(* Logix 5000 project; controller PRU vendor 1 type 14 code 107 rev 20.13; software revision 20.01; part 9 of 17 *)
(* tags used below, declared in another part *)
   AFI : BOOL;
   COOL_FOR_MOTOR_STOP : BOOL;
   CR0_CON1_HTR1_GON : BOOL;   // ZONE 1 (L1,L2,L3)
   CR0_CON1_HTR1_LON : BOOL;   // AUTO LOGIC - ZONE 1 HEATER CONTACTOR
   CR1_CON2_HTR2_GON : BOOL;   // ZONE 2 (L1,L2,L3)
   CR1_CON2_HTR2_LON : BOOL;   // AUTO LOGIC - ZONE 2 HEATER CONTACTOR
   CR2_CON3_HTR3_GON : BOOL;   // ZONE 3 (L1,L2,L3)
   CR2_CON3_HTR3_LON : BOOL;   // AUTO LOGIC - ZONE 3 HEATER CONTACTOR
   CR3_CON4_HTR4_GON : BOOL;   // ZONE 4 (L1) ZONE 5 (L2) ZONE 6 (L3)
   CR3_CON4_HTR4_LON : BOOL;   // AUTO LOGIC - ZONES 4-6 HEATER CONTACTOR
   CR4_CON5_HTR5_GON : BOOL;   // ZONE 7 (L1) ZONE 8 (L2) ZONE 9 (L3)
   CR4_CON5_HTR5_LON : BOOL;   // AUTO LOGIC - ZONES 7-9 HEATER CONTACTOR
   CYCLE_ION_DELAY1_TON : TIMER;
   CYCLE_ION_DELAY2_TON : TIMER;
   CYCLE_ION_DELAY3_TON : TIMER;
   CYCLE_ION_DELAY4_TON : TIMER;
   CYCLE_START_ONS : BOOL;
   CYCLE_START_SS : BOOL;   // Begin temperature ramp and hold heat cycle.
   FAULT : DINT[100];
   FAULT_TIMER : TIMER[10000];
   FAULTS_FA6_IOK : BOOL;   // HEATER FAULTS ARE OK.
   FAULTS_FA6A_IOK : BOOL;
   FAULTS_FA6B_IOK : BOOL;
   HEATER_1_ALARM_ION : BOOL;
   HEATER_2_ALARM_ION : BOOL;
   HEATER_3_ALARM_ION : BOOL;
   HEATER_4_ALARM_ION : BOOL;
   HEATER_5_ALARM_ION : BOOL;
   HEATER_FAULTS_IOK : BOOL;   // FA1, FA4, FA6
   HEATERS_CYCLE_ION : BOOL;   // Heaters are commanded on.
   HMI_ALARM_RESET : BOOL;
   HMI_CYCLE_STOP_PB_ION : BOOL;
   HMI_HEATER_START_PB_ION : BOOL;
   HMI_SEQ_1_FINAL_SETPOINT : DINT;
   HMI_SEQ_1_HOLD_TIME : DINT;
   HMI_SEQ_1_RATE : DINT;
   HMI_SEQ_2_FINAL_SETPOINT : DINT;
   HMI_SEQ_2_HOLD_TIME : DINT;
   HMI_SEQ_2_RATE : DINT;
   HMI_SEQ_3_FINAL_SETPOINT : DINT;
   HMI_SEQ_3_HOLD_TIME : DINT;
   HMI_SEQ_3_RATE : DINT;
   HMI_ZONE1_FINAL_SETPOINT : REAL;
   HMI_ZONE2_FINAL_SETPOINT : DINT;
   HMI_ZONE3_FINAL_SETPOINT : DINT;
   HMI_ZONE4_FINAL_SETPOINT : DINT;
   HMI_ZONE5_FINAL_SETPOINT : REAL;
   HMI_ZONE6_FINAL_SETPOINT : REAL;
   HMI_ZONE7_FINAL_SETPOINT : DINT;
   HMI_ZONE8_FINAL_SETPOINT : DINT;
   HMI_ZONE9_FINAL_SETPOINT : DINT;
   ONE_SEC_SS : BOOL;
   PID_ZONE_1_SETPOINT : DINT;
   PID_ZONE_2_SETPOINT : DINT;
   PID_ZONE_3_SETPOINT : DINT;
   PID_ZONE_4_SETPOINT : DINT;
   PID_ZONE_5_SETPOINT : REAL;
   PID_ZONE_6_SETPOINT : REAL;
   PID_ZONE_7_SETPOINT : DINT;
   PID_ZONE_8_SETPOINT : DINT;
   PID_ZONE_9_SETPOINT : DINT;
   PROCESS_SEQUENCER : INT;
   PRODUCTION_ION : BOOL;
   SEQ_1_HOLD_REM : REAL;
   SEQ_1_HOLD_REM_MIN : REAL;
   SEQ_1_HOLD_TIME : DINT;
   SEQ_1_HOLD_TON : TIMER;
   SEQ_1_HOLDING_ION : BOOL;
   SEQ_1_ION : BOOL;
   SEQ_2_HOLD_REM : REAL;
   SEQ_2_HOLD_REM_MIN : REAL;
   SEQ_2_HOLD_TIME : DINT;
   SEQ_2_HOLD_TON : TIMER;
   SEQ_2_HOLDING_ION : BOOL;
   SEQ_2_ION : BOOL;
   SEQ_3_HOLD_REM : REAL;
   SEQ_3_HOLD_REM_MIN : REAL;
   SEQ_3_HOLD_TIME : DINT;
   SEQ_3_HOLD_TON : TIMER;
   SEQ_3_HOLDING_ION : BOOL;
   SEQ_3_ION : BOOL;
   SEQ_RATE : REAL;
   SP_RATIO : REAL;
   SYSTEM_SETPOINT : REAL;
   TE0101 : REAL;
   TE0102 : REAL;
   TE0103 : REAL;
   TE0104 : REAL;
   TE0105 : REAL;
   TE0106 : REAL;
   TE0107 : REAL;
   TE0108 : REAL;
   TE0109 : REAL;
   TE0110 : REAL;
   TE0111 : REAL;
   TE0112 : REAL;
   TE0113 : REAL;
   TE0114 : REAL;
   TE0115 : REAL;
   TE0116 : REAL;
   TE0117 : REAL;
   TE0118 : REAL;
   TE0119 : REAL;
   TE0120 : REAL;
   TE0121 : REAL;
   TE0122 : REAL;
   TE0123 : REAL;
   TE0124 : REAL;
   TEMP_ZONE_1_AVE : REAL;
   TEMPERATURE_SETPOINT_IS_RAMPING : BOOL;
   TEST_VFD_BON : BOOL;
   THRESHOLD : REAL[9000];
   VFD_SHUTDOWN_TEMP : DINT;
   VFDS_BON : BOOL;   // DRYER VFDs HAVE BEEN COMMANDED ON FOR 1 SECOND.
   Z1_L1_AMPS : REAL;
   Z1_L2_AMPS : REAL;
   Z1_L3_AMPS : REAL;
   Z2_L1_AMPS : REAL;
   Z2_L2_AMPS : REAL;
   Z2_L3_AMPS : REAL;
   Z3_L1_AMPS : REAL;
   Z3_L2_AMPS : REAL;
   Z3_L3_AMPS : REAL;
   Z4_L1_AMPS : REAL;
   Z5_L2_AMPS : REAL;
   Z6_L3_AMPS : REAL;
   Z7_L1_AMPS : REAL;
   Z8_L2_AMPS : REAL;
   Z9_L3_AMPS : REAL;
   ZONE_1_TEMP_AVE : DINT;
(* MainProgram, continued *)

ROUTINE B06_FAULTS_FA6_A_HEATER_5800   (* ladder *)
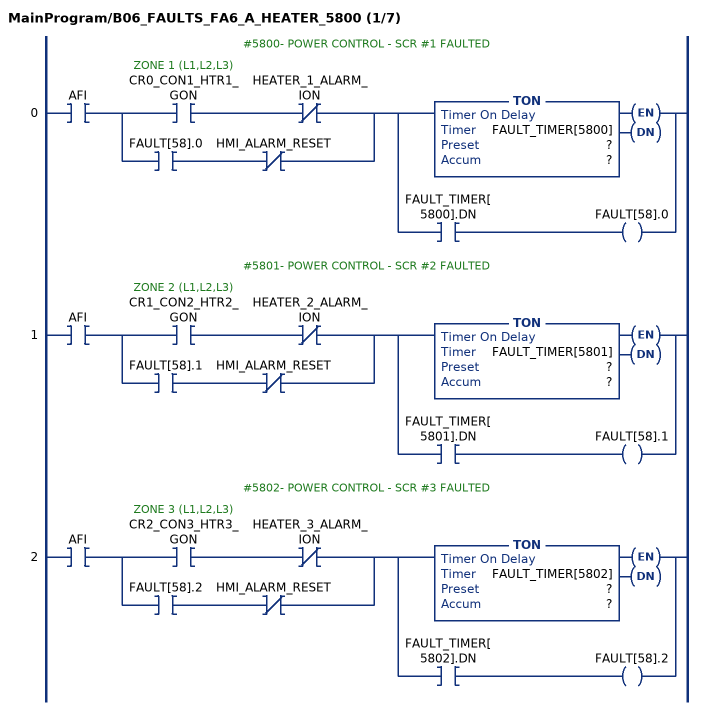
   // #5800- POWER CONTROL - SCR #1 FAULTED
   0: XIC(AFI)[XIC(CR0_CON1_HTR1_GON) XIO(HEATER_1_ALARM_ION) ,XIC(FAULT[58].0) XIO(HMI_ALARM_RESET) ][TON(FAULT_TIMER[5800],?,?) ,XIC(FAULT_TIMER[5800].DN) OTE(FAULT[58].0) ];
   // #5801- POWER CONTROL - SCR #2 FAULTED
   1: XIC(AFI)[XIC(CR1_CON2_HTR2_GON) XIO(HEATER_2_ALARM_ION) ,XIC(FAULT[58].1) XIO(HMI_ALARM_RESET) ][TON(FAULT_TIMER[5801],?,?) ,XIC(FAULT_TIMER[5801].DN) OTE(FAULT[58].1) ];
   // #5802- POWER CONTROL - SCR #3 FAULTED
   2: XIC(AFI)[XIC(CR2_CON3_HTR3_GON) XIO(HEATER_3_ALARM_ION) ,XIC(FAULT[58].2) XIO(HMI_ALARM_RESET) ][TON(FAULT_TIMER[5802],?,?) ,XIC(FAULT_TIMER[5802].DN) OTE(FAULT[58].2) ];
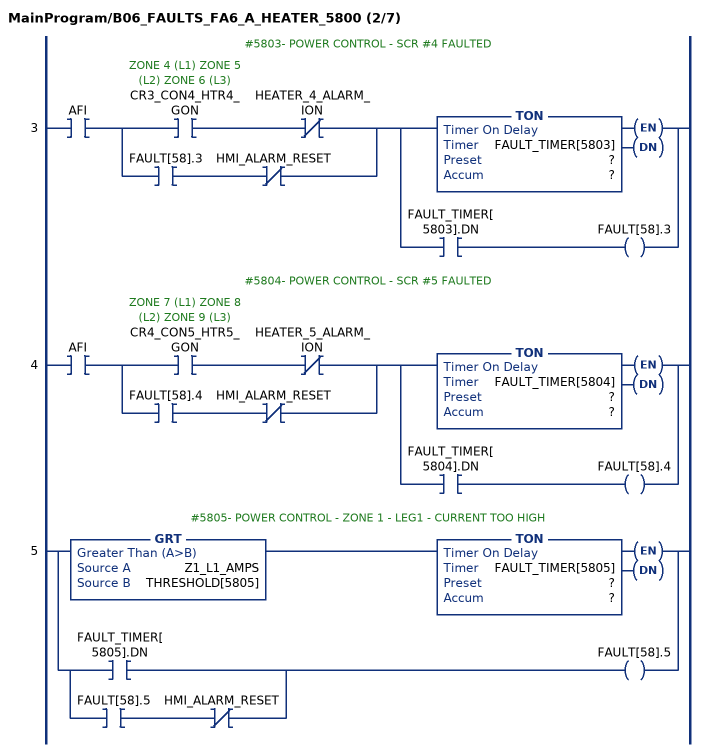
   // #5803- POWER CONTROL - SCR #4 FAULTED
   3: XIC(AFI)[XIC(CR3_CON4_HTR4_GON) XIO(HEATER_4_ALARM_ION) ,XIC(FAULT[58].3) XIO(HMI_ALARM_RESET) ][TON(FAULT_TIMER[5803],?,?) ,XIC(FAULT_TIMER[5803].DN) OTE(FAULT[58].3) ];
   // #5804- POWER CONTROL - SCR #5 FAULTED
   4: XIC(AFI)[XIC(CR4_CON5_HTR5_GON) XIO(HEATER_5_ALARM_ION) ,XIC(FAULT[58].4) XIO(HMI_ALARM_RESET) ][TON(FAULT_TIMER[5804],?,?) ,XIC(FAULT_TIMER[5804].DN) OTE(FAULT[58].4) ];
   // #5805- POWER CONTROL - ZONE 1 - LEG1 - CURRENT TOO HIGH
   5: [GRT(Z1_L1_AMPS,THRESHOLD[5805]) TON(FAULT_TIMER[5805],?,?) ,[XIC(FAULT_TIMER[5805].DN) ,XIC(FAULT[58].5) XIO(HMI_ALARM_RESET) ] OTE(FAULT[58].5) ];
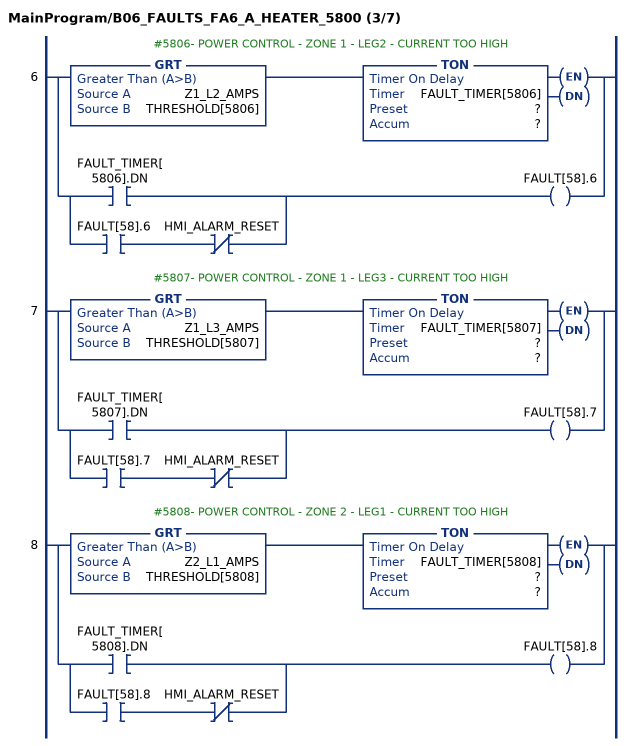
   // #5806- POWER CONTROL - ZONE 1 - LEG2 - CURRENT TOO HIGH
   6: [GRT(Z1_L2_AMPS,THRESHOLD[5806]) TON(FAULT_TIMER[5806],?,?) ,[XIC(FAULT_TIMER[5806].DN) ,XIC(FAULT[58].6) XIO(HMI_ALARM_RESET) ] OTE(FAULT[58].6) ];
   // #5807- POWER CONTROL - ZONE 1 - LEG3 - CURRENT TOO HIGH
   7: [GRT(Z1_L3_AMPS,THRESHOLD[5807]) TON(FAULT_TIMER[5807],?,?) ,[XIC(FAULT_TIMER[5807].DN) ,XIC(FAULT[58].7) XIO(HMI_ALARM_RESET) ] OTE(FAULT[58].7) ];
   // #5808- POWER CONTROL - ZONE 2 - LEG1 - CURRENT TOO HIGH
   8: [GRT(Z2_L1_AMPS,THRESHOLD[5808]) TON(FAULT_TIMER[5808],?,?) ,[XIC(FAULT_TIMER[5808].DN) ,XIC(FAULT[58].8) XIO(HMI_ALARM_RESET) ] OTE(FAULT[58].8) ];
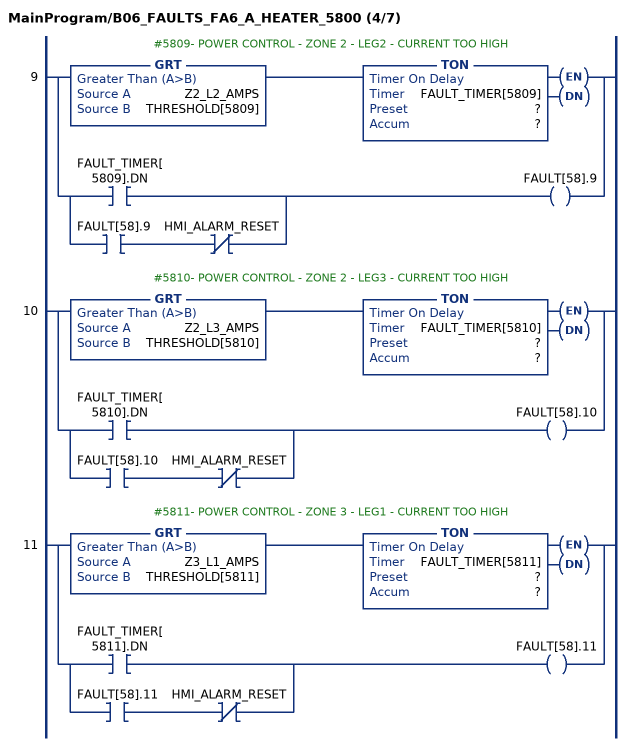
   // #5809- POWER CONTROL - ZONE 2 - LEG2 - CURRENT TOO HIGH
   9: [GRT(Z2_L2_AMPS,THRESHOLD[5809]) TON(FAULT_TIMER[5809],?,?) ,[XIC(FAULT_TIMER[5809].DN) ,XIC(FAULT[58].9) XIO(HMI_ALARM_RESET) ] OTE(FAULT[58].9) ];
   // #5810- POWER CONTROL - ZONE 2 - LEG3 - CURRENT TOO HIGH
   10: [GRT(Z2_L3_AMPS,THRESHOLD[5810]) TON(FAULT_TIMER[5810],?,?) ,[XIC(FAULT_TIMER[5810].DN) ,XIC(FAULT[58].10) XIO(HMI_ALARM_RESET) ] OTE(FAULT[58].10) ];
   // #5811- POWER CONTROL - ZONE 3 - LEG1 - CURRENT TOO HIGH
   11: [GRT(Z3_L1_AMPS,THRESHOLD[5811]) TON(FAULT_TIMER[5811],?,?) ,[XIC(FAULT_TIMER[5811].DN) ,XIC(FAULT[58].11) XIO(HMI_ALARM_RESET) ] OTE(FAULT[58].11) ];
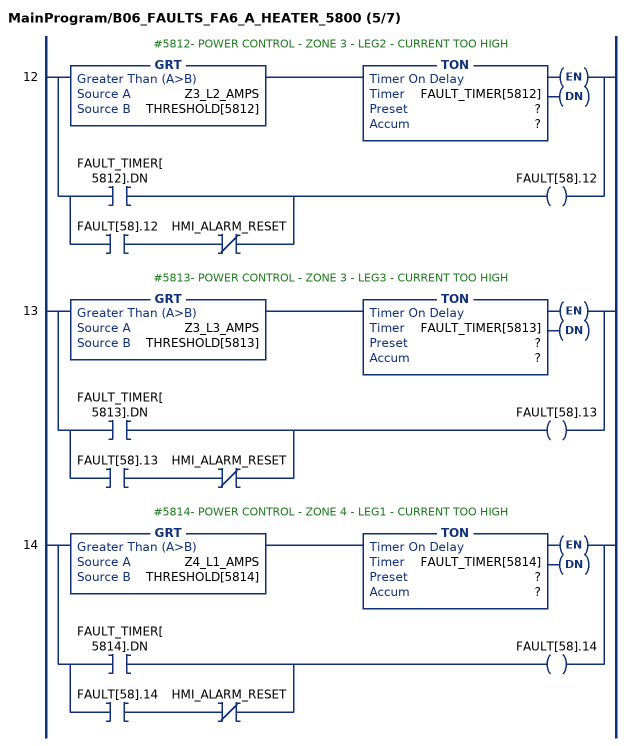
   // #5812- POWER CONTROL - ZONE 3 - LEG2 - CURRENT TOO HIGH
   12: [GRT(Z3_L2_AMPS,THRESHOLD[5812]) TON(FAULT_TIMER[5812],?,?) ,[XIC(FAULT_TIMER[5812].DN) ,XIC(FAULT[58].12) XIO(HMI_ALARM_RESET) ] OTE(FAULT[58].12) ];
   // #5813- POWER CONTROL - ZONE 3 - LEG3 - CURRENT TOO HIGH
   13: [GRT(Z3_L3_AMPS,THRESHOLD[5813]) TON(FAULT_TIMER[5813],?,?) ,[XIC(FAULT_TIMER[5813].DN) ,XIC(FAULT[58].13) XIO(HMI_ALARM_RESET) ] OTE(FAULT[58].13) ];
   // #5814- POWER CONTROL - ZONE 4 - LEG1 - CURRENT TOO HIGH
   14: [GRT(Z4_L1_AMPS,THRESHOLD[5814]) TON(FAULT_TIMER[5814],?,?) ,[XIC(FAULT_TIMER[5814].DN) ,XIC(FAULT[58].14) XIO(HMI_ALARM_RESET) ] OTE(FAULT[58].14) ];
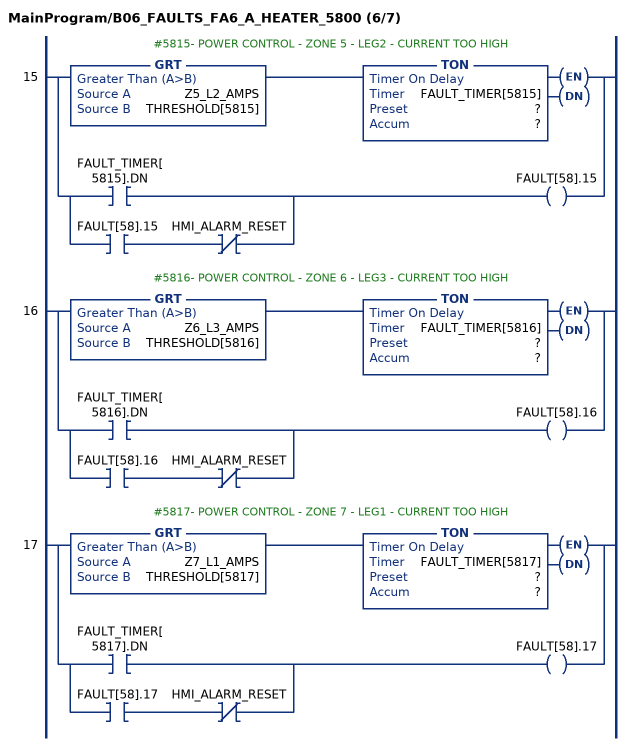
   // #5815- POWER CONTROL - ZONE 5 - LEG2 - CURRENT TOO HIGH
   15: [GRT(Z5_L2_AMPS,THRESHOLD[5815]) TON(FAULT_TIMER[5815],?,?) ,[XIC(FAULT_TIMER[5815].DN) ,XIC(FAULT[58].15) XIO(HMI_ALARM_RESET) ] OTE(FAULT[58].15) ];
   // #5816- POWER CONTROL - ZONE 6 - LEG3 - CURRENT TOO HIGH
   16: [GRT(Z6_L3_AMPS,THRESHOLD[5816]) TON(FAULT_TIMER[5816],?,?) ,[XIC(FAULT_TIMER[5816].DN) ,XIC(FAULT[58].16) XIO(HMI_ALARM_RESET) ] OTE(FAULT[58].16) ];
   // #5817- POWER CONTROL - ZONE 7 - LEG1 - CURRENT TOO HIGH
   17: [GRT(Z7_L1_AMPS,THRESHOLD[5817]) TON(FAULT_TIMER[5817],?,?) ,[XIC(FAULT_TIMER[5817].DN) ,XIC(FAULT[58].17) XIO(HMI_ALARM_RESET) ] OTE(FAULT[58].17) ];
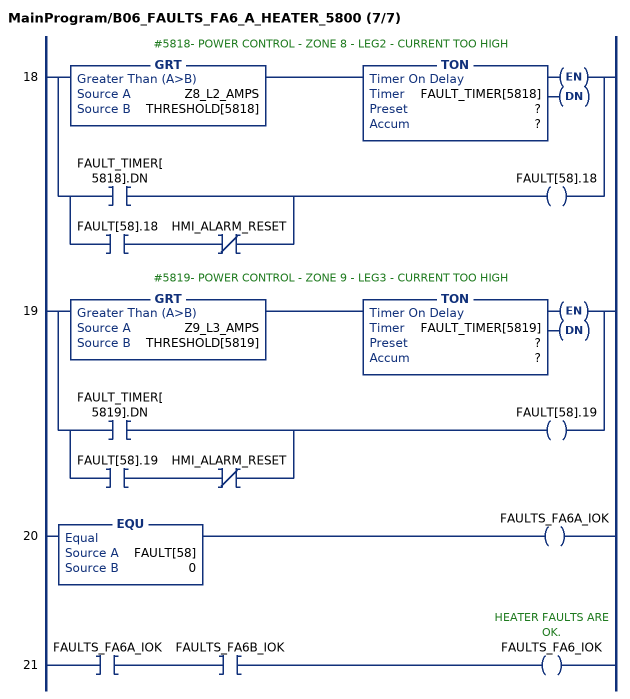
   // #5818- POWER CONTROL - ZONE 8 - LEG2 - CURRENT TOO HIGH
   18: [GRT(Z8_L2_AMPS,THRESHOLD[5818]) TON(FAULT_TIMER[5818],?,?) ,[XIC(FAULT_TIMER[5818].DN) ,XIC(FAULT[58].18) XIO(HMI_ALARM_RESET) ] OTE(FAULT[58].18) ];
   // #5819- POWER CONTROL - ZONE 9 - LEG3 - CURRENT TOO HIGH
   19: [GRT(Z9_L3_AMPS,THRESHOLD[5819]) TON(FAULT_TIMER[5819],?,?) ,[XIC(FAULT_TIMER[5819].DN) ,XIC(FAULT[58].19) XIO(HMI_ALARM_RESET) ] OTE(FAULT[58].19) ];
   20: EQU(FAULT[58],0)OTE(FAULTS_FA6A_IOK);
   21: XIC(FAULTS_FA6A_IOK)XIC(FAULTS_FA6B_IOK)OTE(FAULTS_FA6_IOK);
END_ROUTINE

ROUTINE C00_CYCLE_START   (* ladder *)
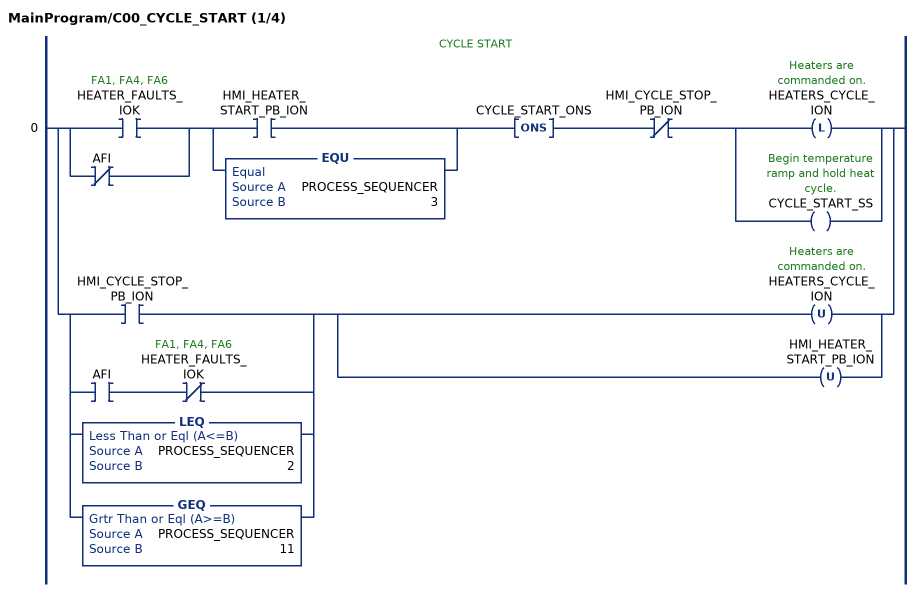
   // CYCLE START
   0: [[XIC(HEATER_FAULTS_IOK) ,XIO(AFI) ] [XIC(HMI_HEATER_START_PB_ION) ,EQU(PROCESS_SEQUENCER,3) ] ONS(CYCLE_START_ONS) XIO(HMI_CYCLE_STOP_PB_ION) [OTL(HEATERS_CYCLE_ION) ,OTE(CYCLE_START_SS) ] ,[XIC(HMI_CYCLE_STOP_PB_ION) ,XIC(AFI) XIO(HEATER_FAULTS_IOK) ,LEQ(PROCESS_SEQUENCER,2) ,GEQ(PROCESS_SEQUENCER,11) ] [OTU(HEATERS_CYCLE_ION) ,OTU(HMI_HEATER_START_PB_ION) ] ];
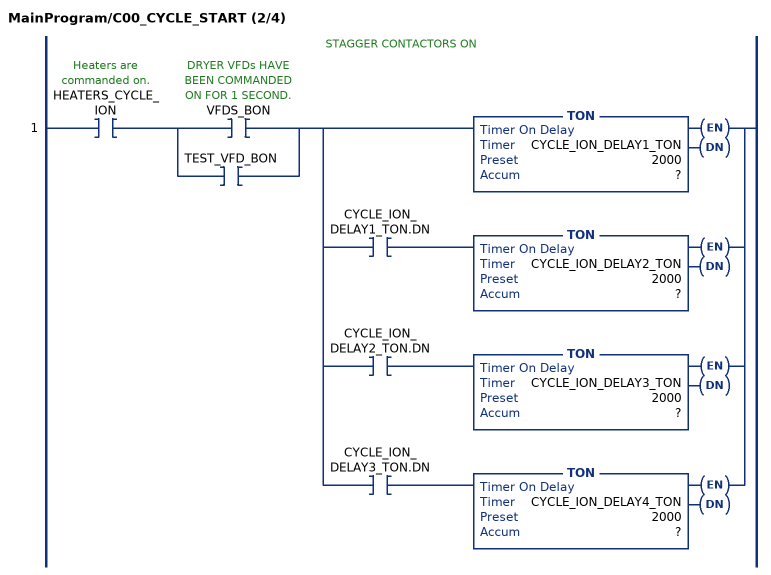
   // STAGGER CONTACTORS ON
   1: XIC(HEATERS_CYCLE_ION)[XIC(VFDS_BON) ,XIC(TEST_VFD_BON) ][TON(CYCLE_ION_DELAY1_TON,?,?) ,XIC(CYCLE_ION_DELAY1_TON.DN) TON(CYCLE_ION_DELAY2_TON,?,?) ,XIC(CYCLE_ION_DELAY2_TON.DN) TON(CYCLE_ION_DELAY3_TON,?,?) ,XIC(CYCLE_ION_DELAY3_TON.DN) TON(CYCLE_ION_DELAY4_TON,?,?) ];
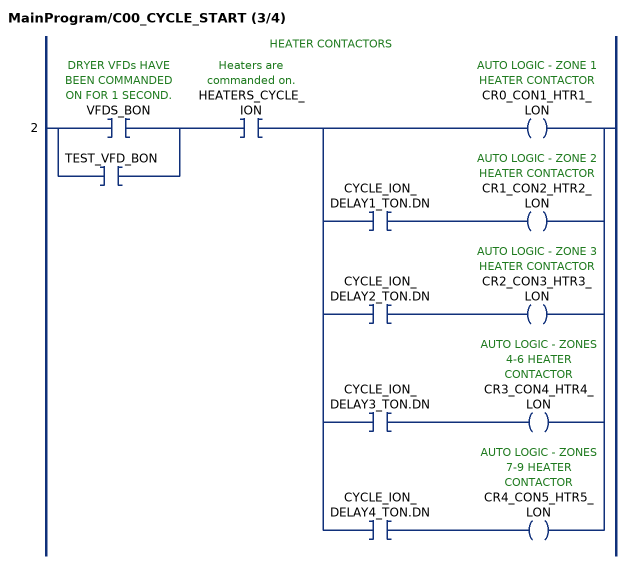
   // HEATER CONTACTORS
   2: [XIC(VFDS_BON) ,XIC(TEST_VFD_BON) ]XIC(HEATERS_CYCLE_ION)[OTE(CR0_CON1_HTR1_LON) ,XIC(CYCLE_ION_DELAY1_TON.DN) OTE(CR1_CON2_HTR2_LON) ,XIC(CYCLE_ION_DELAY2_TON.DN) OTE(CR2_CON3_HTR3_LON) ,XIC(CYCLE_ION_DELAY3_TON.DN) OTE(CR3_CON4_HTR4_LON) ,XIC(CYCLE_ION_DELAY4_TON.DN) OTE(CR4_CON5_HTR5_LON) ];
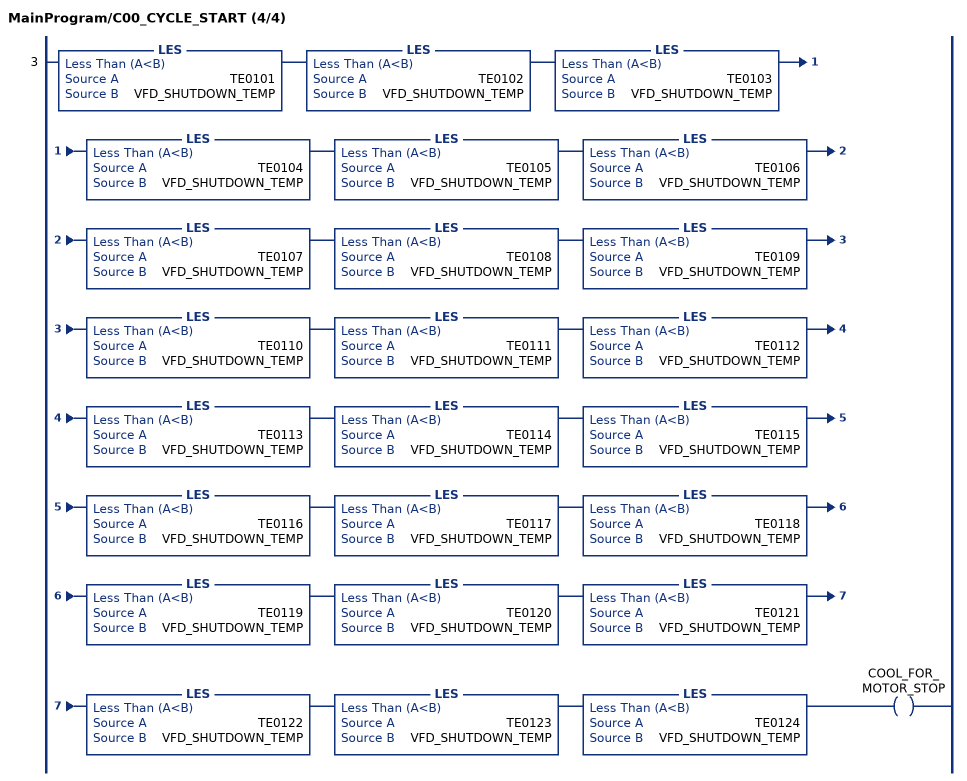
   3: LES(TE0101,VFD_SHUTDOWN_TEMP)LES(TE0102,VFD_SHUTDOWN_TEMP)LES(TE0103,VFD_SHUTDOWN_TEMP)LES(TE0104,VFD_SHUTDOWN_TEMP)LES(TE0105,VFD_SHUTDOWN_TEMP)LES(TE0106,VFD_SHUTDOWN_TEMP)LES(TE0107,VFD_SHUTDOWN_TEMP)LES(TE0108,VFD_SHUTDOWN_TEMP)LES(TE0109,VFD_SHUTDOWN_TEMP)LES(TE0110,VFD_SHUTDOWN_TEMP)LES(TE0111,VFD_SHUTDOWN_TEMP)LES(TE0112,VFD_SHUTDOWN_TEMP)LES(TE0113,VFD_SHUTDOWN_TEMP)LES(TE0114,VFD_SHUTDOWN_TEMP)LES(TE0115,VFD_SHUTDOWN_TEMP)LES(TE0116,VFD_SHUTDOWN_TEMP)LES(TE0117,VFD_SHUTDOWN_TEMP)LES(TE0118,VFD_SHUTDOWN_TEMP)LES(TE0119,VFD_SHUTDOWN_TEMP)LES(TE0120,VFD_SHUTDOWN_TEMP)LES(TE0121,VFD_SHUTDOWN_TEMP)LES(TE0122,VFD_SHUTDOWN_TEMP)LES(TE0123,VFD_SHUTDOWN_TEMP)LES(TE0124,VFD_SHUTDOWN_TEMP)OTE(COOL_FOR_MOTOR_STOP);
END_ROUTINE

ROUTINE C01_CYCLE_SEQUENCES   (* ladder *)
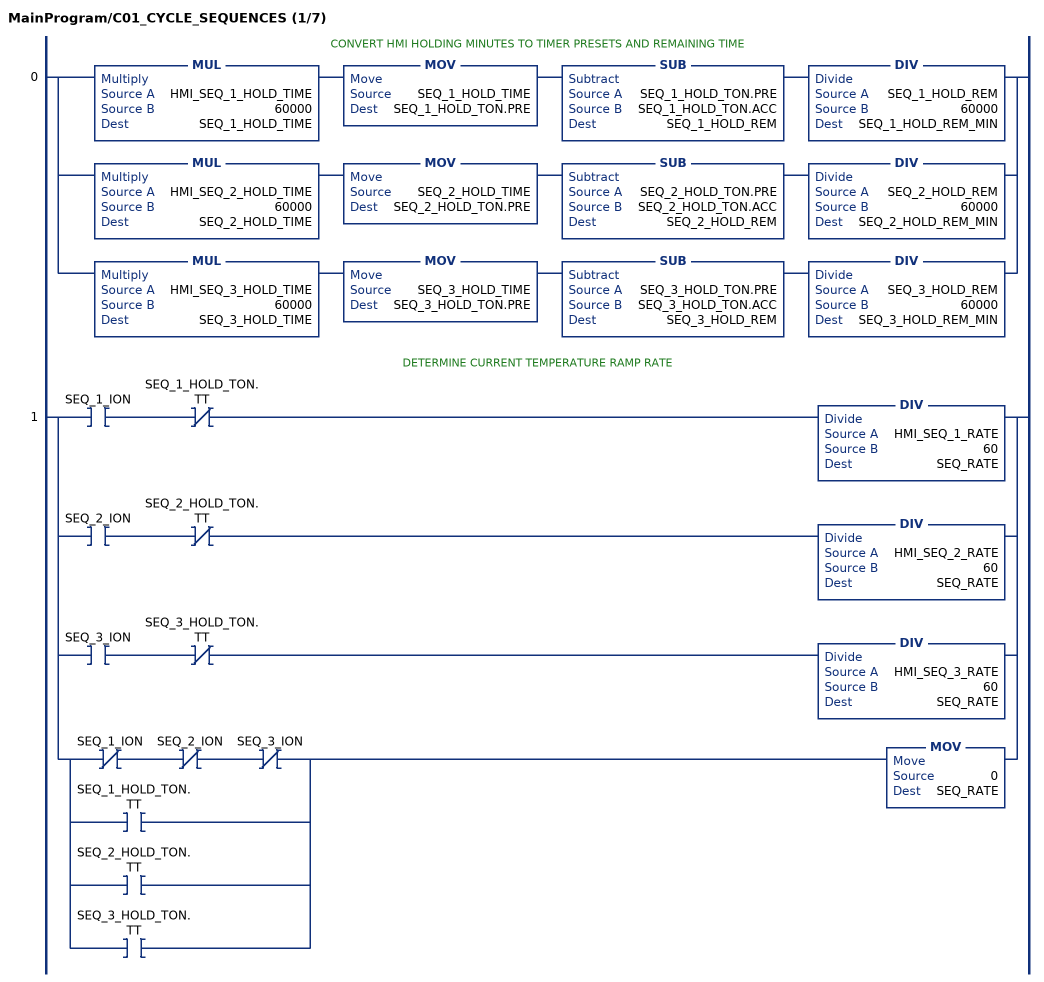
   // CONVERT HMI HOLDING MINUTES TO TIMER PRESETS AND REMAINING TIME
   0: [MUL(HMI_SEQ_1_HOLD_TIME,60000,SEQ_1_HOLD_TIME) MOV(SEQ_1_HOLD_TIME,SEQ_1_HOLD_TON.PRE) SUB(SEQ_1_HOLD_TON.PRE,SEQ_1_HOLD_TON.ACC,SEQ_1_HOLD_REM) DIV(SEQ_1_HOLD_REM,60000,SEQ_1_HOLD_REM_MIN) ,MUL(HMI_SEQ_2_HOLD_TIME,60000,SEQ_2_HOLD_TIME) MOV(SEQ_2_HOLD_TIME,SEQ_2_HOLD_TON.PRE) SUB(SEQ_2_HOLD_TON.PRE,SEQ_2_HOLD_TON.ACC,SEQ_2_HOLD_REM) DIV(SEQ_2_HOLD_REM,60000,SEQ_2_HOLD_REM_MIN) ,MUL(HMI_SEQ_3_HOLD_TIME,60000,SEQ_3_HOLD_TIME) MOV(SEQ_3_HOLD_TIME,SEQ_3_HOLD_TON.PRE) SUB(SEQ_3_HOLD_TON.PRE,SEQ_3_HOLD_TON.ACC,SEQ_3_HOLD_REM) DIV(SEQ_3_HOLD_REM,60000,SEQ_3_HOLD_REM_MIN) ];
   // DETERMINE CURRENT TEMPERATURE RAMP RATE
   1: [XIC(SEQ_1_ION) XIO(SEQ_1_HOLD_TON.TT) DIV(HMI_SEQ_1_RATE,60,SEQ_RATE) ,XIC(SEQ_2_ION) XIO(SEQ_2_HOLD_TON.TT) DIV(HMI_SEQ_2_RATE,60,SEQ_RATE) ,XIC(SEQ_3_ION) XIO(SEQ_3_HOLD_TON.TT) DIV(HMI_SEQ_3_RATE,60,SEQ_RATE) ,[XIO(SEQ_1_ION) XIO(SEQ_2_ION) XIO(SEQ_3_ION) ,XIC(SEQ_1_HOLD_TON.TT) ,XIC(SEQ_2_HOLD_TON.TT) ,XIC(SEQ_3_HOLD_TON.TT) ] MOV(0,SEQ_RATE) ];
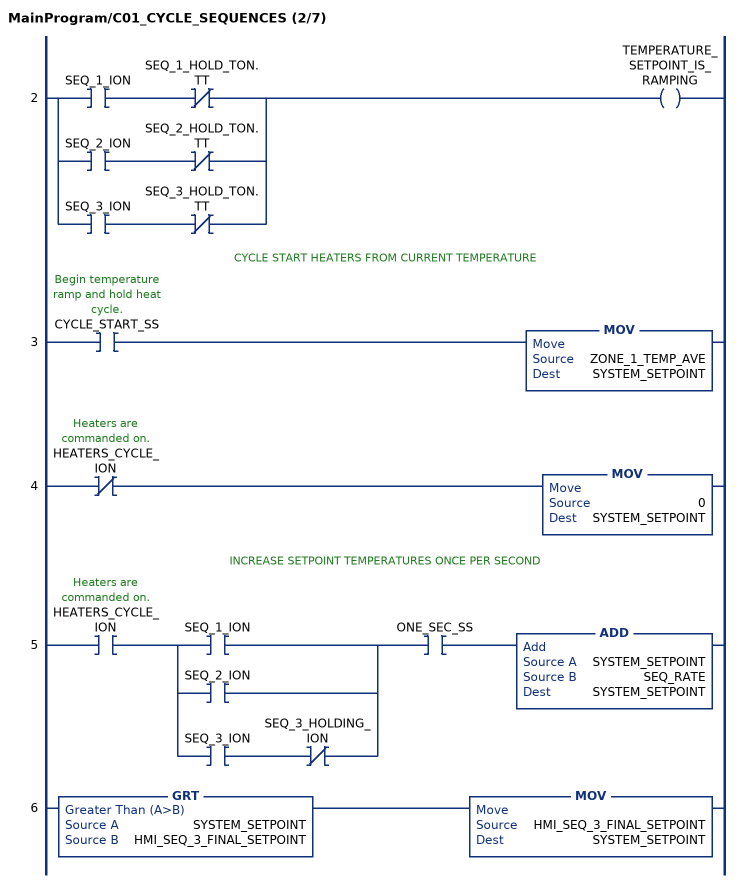
   2: [XIC(SEQ_1_ION) XIO(SEQ_1_HOLD_TON.TT) ,XIC(SEQ_2_ION) XIO(SEQ_2_HOLD_TON.TT) ,XIC(SEQ_3_ION) XIO(SEQ_3_HOLD_TON.TT) ]OTE(TEMPERATURE_SETPOINT_IS_RAMPING);
   // CYCLE START HEATERS FROM CURRENT TEMPERATURE
   3: XIC(CYCLE_START_SS)MOV(ZONE_1_TEMP_AVE,SYSTEM_SETPOINT);
   4: XIO(HEATERS_CYCLE_ION)MOV(0,SYSTEM_SETPOINT);
   // INCREASE SETPOINT TEMPERATURES ONCE PER SECOND
   5: XIC(HEATERS_CYCLE_ION)[XIC(SEQ_1_ION) ,XIC(SEQ_2_ION) ,XIC(SEQ_3_ION) XIO(SEQ_3_HOLDING_ION) ]XIC(ONE_SEC_SS)ADD(SYSTEM_SETPOINT,SEQ_RATE,SYSTEM_SETPOINT);
   6: GRT(SYSTEM_SETPOINT,HMI_SEQ_3_FINAL_SETPOINT)MOV(HMI_SEQ_3_FINAL_SETPOINT,SYSTEM_SETPOINT);
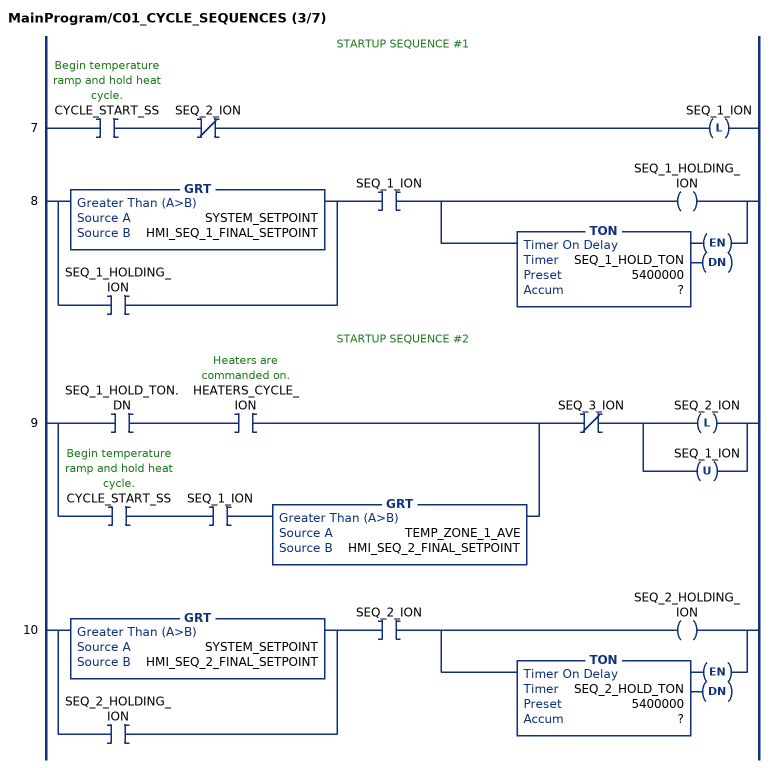
   // STARTUP SEQUENCE #1
   7: XIC(CYCLE_START_SS)XIO(SEQ_2_ION)OTL(SEQ_1_ION);
   8: [GRT(SYSTEM_SETPOINT,HMI_SEQ_1_FINAL_SETPOINT) ,XIC(SEQ_1_HOLDING_ION) ]XIC(SEQ_1_ION)[OTE(SEQ_1_HOLDING_ION) ,TON(SEQ_1_HOLD_TON,?,?) ];
   // STARTUP SEQUENCE #2
   9: [XIC(SEQ_1_HOLD_TON.DN) XIC(HEATERS_CYCLE_ION) ,XIC(CYCLE_START_SS) XIC(SEQ_1_ION) GRT(TEMP_ZONE_1_AVE,HMI_SEQ_2_FINAL_SETPOINT) ]XIO(SEQ_3_ION)[OTL(SEQ_2_ION) ,OTU(SEQ_1_ION) ];
   10: [GRT(SYSTEM_SETPOINT,HMI_SEQ_2_FINAL_SETPOINT) ,XIC(SEQ_2_HOLDING_ION) ]XIC(SEQ_2_ION)[OTE(SEQ_2_HOLDING_ION) ,TON(SEQ_2_HOLD_TON,?,?) ];
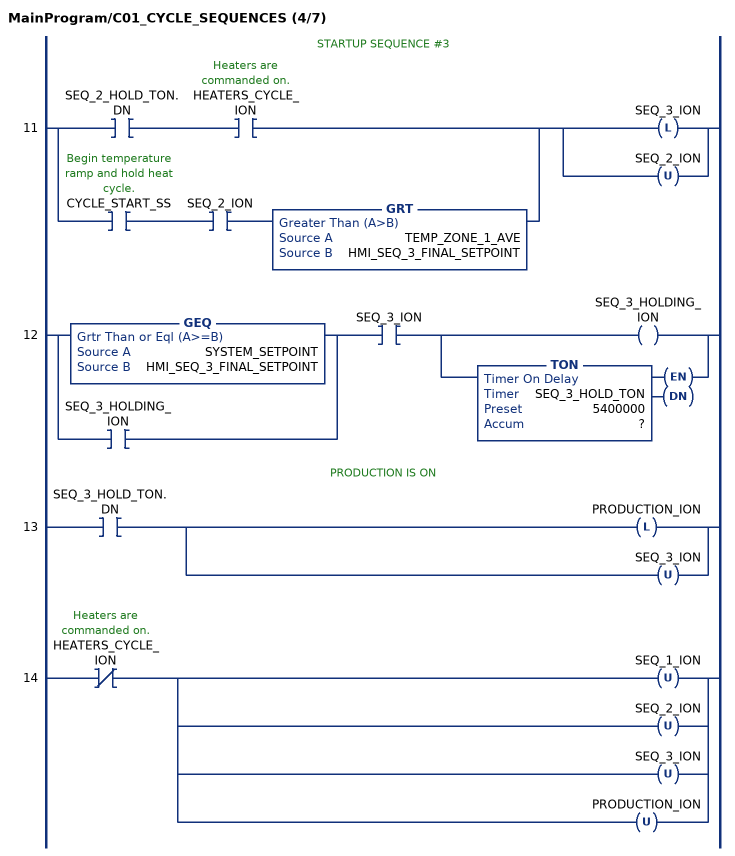
   // STARTUP SEQUENCE #3
   11: [XIC(SEQ_2_HOLD_TON.DN) XIC(HEATERS_CYCLE_ION) ,XIC(CYCLE_START_SS) XIC(SEQ_2_ION) GRT(TEMP_ZONE_1_AVE,HMI_SEQ_3_FINAL_SETPOINT) ][OTL(SEQ_3_ION) ,OTU(SEQ_2_ION) ];
   12: [GEQ(SYSTEM_SETPOINT,HMI_SEQ_3_FINAL_SETPOINT) ,XIC(SEQ_3_HOLDING_ION) ]XIC(SEQ_3_ION)[OTE(SEQ_3_HOLDING_ION) ,TON(SEQ_3_HOLD_TON,?,?) ];
   // PRODUCTION IS ON
   13: XIC(SEQ_3_HOLD_TON.DN)[OTL(PRODUCTION_ION) ,OTU(SEQ_3_ION) ];
   14: XIO(HEATERS_CYCLE_ION)[OTU(SEQ_1_ION) ,OTU(SEQ_2_ION) ,OTU(SEQ_3_ION) ,OTU(PRODUCTION_ION) ];
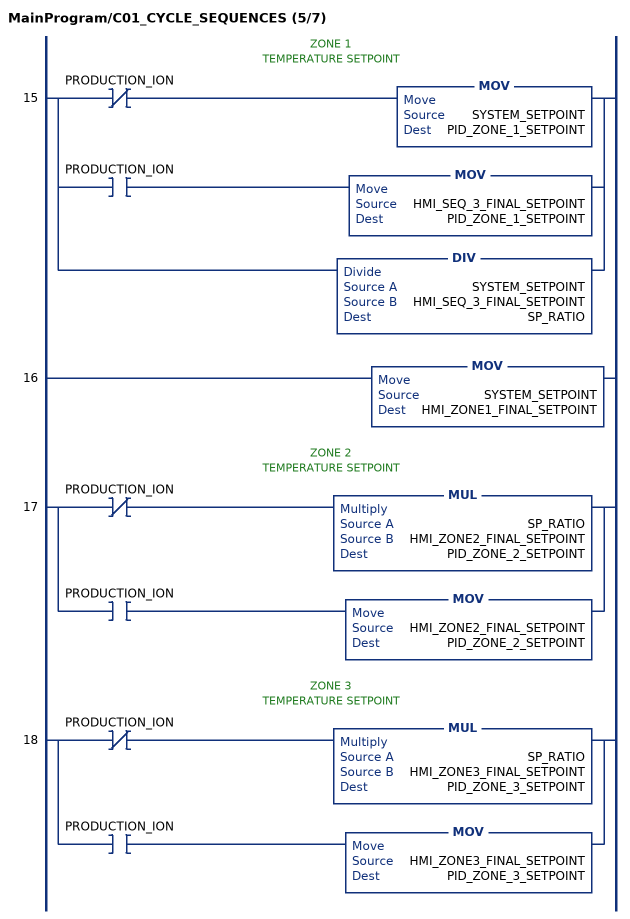
   // ZONE 1
   // TEMPERATURE SETPOINT
   15: [XIO(PRODUCTION_ION) MOV(SYSTEM_SETPOINT,PID_ZONE_1_SETPOINT) ,XIC(PRODUCTION_ION) MOV(HMI_SEQ_3_FINAL_SETPOINT,PID_ZONE_1_SETPOINT) ,DIV(SYSTEM_SETPOINT,HMI_SEQ_3_FINAL_SETPOINT,SP_RATIO) ];
   16: MOV(SYSTEM_SETPOINT,HMI_ZONE1_FINAL_SETPOINT);
   // ZONE 2
   // TEMPERATURE SETPOINT
   17: [XIO(PRODUCTION_ION) MUL(SP_RATIO,HMI_ZONE2_FINAL_SETPOINT,PID_ZONE_2_SETPOINT) ,XIC(PRODUCTION_ION) MOV(HMI_ZONE2_FINAL_SETPOINT,PID_ZONE_2_SETPOINT) ];
   // ZONE 3
   // TEMPERATURE SETPOINT
   18: [XIO(PRODUCTION_ION) MUL(SP_RATIO,HMI_ZONE3_FINAL_SETPOINT,PID_ZONE_3_SETPOINT) ,XIC(PRODUCTION_ION) MOV(HMI_ZONE3_FINAL_SETPOINT,PID_ZONE_3_SETPOINT) ];
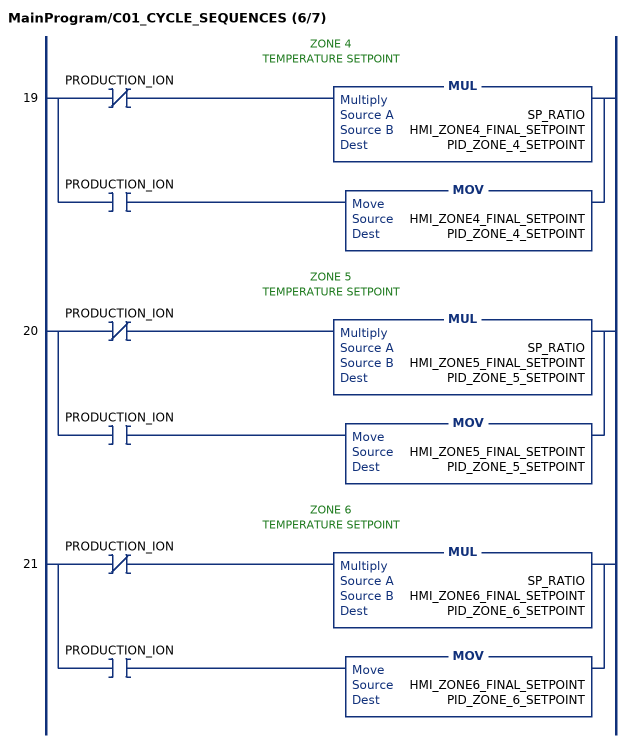
   // ZONE 4
   // TEMPERATURE SETPOINT
   19: [XIO(PRODUCTION_ION) MUL(SP_RATIO,HMI_ZONE4_FINAL_SETPOINT,PID_ZONE_4_SETPOINT) ,XIC(PRODUCTION_ION) MOV(HMI_ZONE4_FINAL_SETPOINT,PID_ZONE_4_SETPOINT) ];
   // ZONE 5
   // TEMPERATURE SETPOINT
   20: [XIO(PRODUCTION_ION) MUL(SP_RATIO,HMI_ZONE5_FINAL_SETPOINT,PID_ZONE_5_SETPOINT) ,XIC(PRODUCTION_ION) MOV(HMI_ZONE5_FINAL_SETPOINT,PID_ZONE_5_SETPOINT) ];
   // ZONE 6
   // TEMPERATURE SETPOINT
   21: [XIO(PRODUCTION_ION) MUL(SP_RATIO,HMI_ZONE6_FINAL_SETPOINT,PID_ZONE_6_SETPOINT) ,XIC(PRODUCTION_ION) MOV(HMI_ZONE6_FINAL_SETPOINT,PID_ZONE_6_SETPOINT) ];
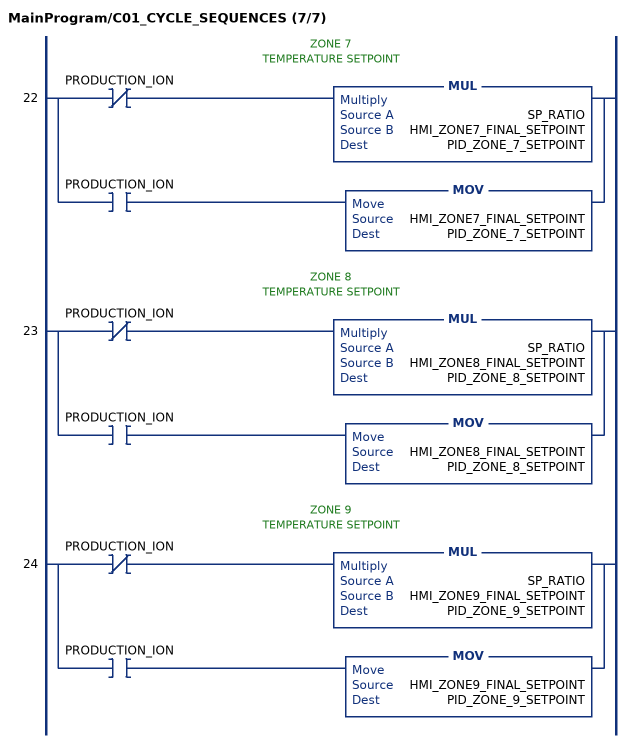
   // ZONE 7
   // TEMPERATURE SETPOINT
   22: [XIO(PRODUCTION_ION) MUL(SP_RATIO,HMI_ZONE7_FINAL_SETPOINT,PID_ZONE_7_SETPOINT) ,XIC(PRODUCTION_ION) MOV(HMI_ZONE7_FINAL_SETPOINT,PID_ZONE_7_SETPOINT) ];
   // ZONE 8
   // TEMPERATURE SETPOINT
   23: [XIO(PRODUCTION_ION) MUL(SP_RATIO,HMI_ZONE8_FINAL_SETPOINT,PID_ZONE_8_SETPOINT) ,XIC(PRODUCTION_ION) MOV(HMI_ZONE8_FINAL_SETPOINT,PID_ZONE_8_SETPOINT) ];
   // ZONE 9
   // TEMPERATURE SETPOINT
   24: [XIO(PRODUCTION_ION) MUL(SP_RATIO,HMI_ZONE9_FINAL_SETPOINT,PID_ZONE_9_SETPOINT) ,XIC(PRODUCTION_ION) MOV(HMI_ZONE9_FINAL_SETPOINT,PID_ZONE_9_SETPOINT) ];
END_ROUTINE
